// TwinCAT 3 PLC project PLC1
// ProgramVersion: 3.1.4026.22
// libraries:
//   Tc2_EtherCAT, * (Beckhoff Automation GmbH)
//   Tc2_Standard, * (Beckhoff Automation GmbH)
//   Tc2_System, * (Beckhoff Automation GmbH)
//   Tc3_RealtimeMonitoring, * (Beckhoff Automation GmbH)
// project tree:
//   GVLs/ FB_DoWork.TcPOU (not stored), GVL.TcGVL
//   POUs/ F_ConsumeTime.TcPOU, PRG_Task1.TcPOU, PRG_Task2.TcPOU, PRG_Task3.TcPOU
//   / Task1.TcTTO (not stored), Task2.TcTTO (not stored), Task3.TcTTO

CONFIGURATION PLC1
    RESOURCE PLC ON TwinCAT3
        TASK Task3(INTERVAL := T#10ms, PRIORITY := 13);
        PROGRAM PRG_Task3 WITH Task3 : PRG_Task3;
    END_RESOURCE
END_CONFIGURATION

// ---- GVLs/GVL.TcGVL
{attribute 'qualified_only'}
VAR_GLOBAL
	bGlobalTestFlag : BOOL;
	fbDoWork		: FB_DoWork;
END_VAR

// ---- POUs/PRG_Task3.TcPOU
PROGRAM PRG_Task3
VAR
	{attribute 'displaymode':='hex'}
	CallingTaskAdsPort	 : UINT;
	nLocalBlockedCounter : DINT;
END_VAR

CallingTaskAdsPort := _TaskInfo[GETCURTASKINDEXEX()].AdsPort;
WHILE NOT (TestAndSet(GVL.bGlobalTestFlag)) DO //Spin
	nLocalBlockedCounter := nLocalBlockedCounter + 1;
END_WHILE

(* bGlobalTestFlag was FALSE, nobody was blocking, NOW
bGlobalTestFlag is set to TRUE and blocking others *)
GVL.fbDoWork.M_ConsumeTime(CallerTaskAdsPort := CallingTaskAdsPort);

(* remove blocking by resetting the flag *)
GVL.bGlobalTestFlag := FALSE;

END_PROGRAM

// ---- POUs/F_ConsumeTime.TcPOU
FUNCTION F_ConsumeTime
VAR_INPUT
	Us		:UDINT;
END_VAR
VAR
		tCurr, tEnd : T_DCTIME64;
END_VAR

tCurr := F_GetActualDcTime64();
tEnd  := tCurr + (Us * EC_DCTIME_TICKSPERMSEC64 / 1000);
WHILE (tCurr < tEnd) DO
	tCurr := F_GetActualDcTime64();
END_WHILE

END_FUNCTION

// ---- POUs/PRG_Task1.TcPOU
PROGRAM PRG_Task1
VAR
	{attribute 'displaymode':='hex'}
	CallingTaskAdsPort	 : UINT;
	nLocalBlockedCounter : DINT;
END_VAR

CallingTaskAdsPort := _TaskInfo[GETCURTASKINDEXEX()].AdsPort;
WHILE NOT (TestAndSet(GVL.bGlobalTestFlag)) DO //Spin
	nLocalBlockedCounter := nLocalBlockedCounter + 1; 
END_WHILE

(* bGlobalTestFlag was FALSE, nobody was blocking, NOW
    bGlobalTestFlag is set to TRUE and blocking others *)
GVL.fbDoWork.M_ConsumeTime(CallerTaskAdsPort := CallingTaskAdsPort);

(* remove blocking by resetting the flag *)
GVL.bGlobalTestFlag := FALSE;

END_PROGRAM

// ---- POUs/PRG_Task2.TcPOU
PROGRAM PRG_Task2
VAR
	//Just another task on the same core as task 1 to show the
	//scedular executing another task if task 1 gets blocked
END_VAR

F_ConsumeTime(400);

END_PROGRAM
